{attribute 'qualified_only'}
VAR_GLOBAL
	TxWord1	: WORD;
	TxWord2 : WORD;
	TxWord3 : WORD;
	
	RxWord1 : WORD;
	RxWord2 : WORD;
	RxWord3 : WORD;

	
	TxInt : ARRAY [1..5] OF INT;
	TxDint : ARRAY [1..3] OF DINT;
	TxREAL : ARRAY [1..7] OF REAL;

	RxInt : ARRAY [1..2] OF INT;
	RxDint : ARRAY [1..3] OF DINT;
	RxREAL : ARRAY [1..44] OF REAL;
	
	Charger : ARRAY[1..7] OF ST_Charger_Base;
	
	TDKLoad	: ARRAY [1..7] OF ST_Setpoints_Base; 
	
	(*ChargerHVOFF_rlyDelayPT		: TIME := T#25MS;
	ChargerHVOFF_rlyDelayPT_INT	: INT := 25;
	
	HVONdelayPT					: TIME := T#250MS;
	HVONdelayPT_INT				: INT := 250;
	
	RunOutTMR_PT				: TIME := T#10S;
	RunOutTMR_PT_INT			: DINT := 10;
	RunOutTMR_elapse			: DINT;
	
	ChargingRunOutTMR_elapse	: INT;
	
	ChargePB					: BOOL := 0;
	DumpPB						: BOOL := 0;
	AbortPB						: BOOL := 0;
	FirePB						: BOOL := 0;
	ClearFaultPB				: BOOL := 0;
	AllDumpRelaysOpenBP			: BOOL := 0;
	AllChargeRelayCloseBP		: BOOL := 0;
	SystemSafeBP				: BOOL := 0;
	
	HMI_ManualModeSelected		: BOOL := 0;  // 1 = manual mode selected
	CloseChargeRlySW			: BOOL := 0;
	OpenDumpRlySW				: BOOL := 0;*)
END_VAR

(* stored: Version 1.1.0.1, ProductVersion 3.1.4024.11
   GVL LV: Id {a1b8c407-04a5-4145-a7ff-e33fdc4ffda1} *)
